// TIA Portal V17 export
// export: Created 2024-01-30T08:49:16.6379613Z, ExportSetting WithDefaults, DisplayName Totally Integrated Automation Portal, DisplayVersion V17 Update 6, DisplayName TIA Portal Openness, DisplayVersion V17 Update 6, DisplayName TIA Portal Version Control Interface, DisplayVersion V17, DisplayName STEP 7 Professional, DisplayVersion V17 Update 6, DisplayName STEP 7 Safety, DisplayVersion V17 Update 6, DisplayName WinCC Advanced, DisplayVersion V17 Update 6
DATA_BLOCK "FFT_BREMEN_SPS_Connection_DB_2"   // DB38
{ S7_Optimized_Access := 'TRUE' }
// stored: AutoNumber true, DBAccessibleFromOPCUA true, DBAccessibleFromWebserver true, InstanceOfName TCON_IP_v4, OfSystemLibElement TCON_IP_v4, OfSystemLibVersion 1.0
"TCON_IP_v4"
   // VAR
   //    InterfaceId : HW_ANY := 64;
   //    ID : CONN_OUC := 3;
   //    ConnectionType : Byte;
   //    ActiveEstablished : Bool := true;
   //    RemoteAddress { S7_SetPoint := 'True'} : IP_V4;
   //    RemotePort : UInt := 2001;
   //    LocalPort : UInt := 2000;
   // END_VAR
BEGIN
   RemoteAddress.ADDR[1] := 10;
   RemoteAddress.ADDR[2] := 183;
   RemoteAddress.ADDR[3] := 122;
   RemoteAddress.ADDR[4] := 3;
END_DATA_BLOCK
